// TIA Portal V18 export
// export: Created 2025-12-01T17:53:01.7250891Z, ExportSetting None, DisplayName Totally Integrated Automation Portal, DisplayVersion V18 Update 5, DisplayName TIA Portal Openness, DisplayVersion V18 Update 5, DisplayName TIA Portal Teamcenter Gateway, DisplayVersion V18, DisplayName TIA Portal Version Control Interface, DisplayVersion V18, DisplayName STEP 7 Professional, DisplayVersion V18 Update 5, DisplayName STEP 7 Safety, DisplayVersion V18, DisplayName WinCC Professional, DisplayVersion V18 Update 5
Screen "240_Cylinder_E1"  1280x800, Number=240, Template=02ManualUnit1
  ScreenLayer "Layer_0"
    FaceplateInstance "Cylinder_S71500_TP700_1" at 0,85 size 1279x80  FaceplateTypeName=03 FunctionBlocks@$@101 Cylinder@$@101.2 HMI@$@S7-1500@$@Cylinder_S71500_TP700 V 0.0.29
      Cy := STxxxCylinder011
      CylinderName := Cyl name
      HomeButtonName := Cyl go home button
      WorkButtonName := Cyl go work button
      HomeQaddress := Cyl home Q
      HomeIaddress := Cyl home I
      WorkIaddress := Cyl work I
      WorkQaddress := Cyl work Q
    Button "btnMenu4" at 384,725 size 128x75  StyleItem=BtnNormal20
    Button "btnMenu5" at 512,725 size 128x75  StyleItem=BtnNormal20
    Button "btnMenu6" at 640,725 size 128x75  StyleItem=BtnNormal20
    Button "btnMenu6_1" at 768,725 size 128x75  StyleItem=BtnNormal20
    Button "按钮_1" at 128,725 size 128x75  PictureOff=向右箭头_0, TextOff="E-气缸1 / E-Cylinder1", TextOn="E-气缸1 / E-Cylinder1"
      on Click: ActivateScreen(Screen name := , Object number := 0)
    Button "btnMenu4_1" at 256,725 size 128x75  TextOff="E-气缸2 / E-Cylinder2", TextOn="E-气缸2 / E-Cylinder2"
      on Click: ActivateScreen(Screen name := 246_Cylinder_E2, Object number := 0)
    GraphicView "图形视图_1" at 353,167 size 602x502  Picture=图形_52
    Button "btnMenu7" at 896,725 size 128x75
    Button "btnMenu7_1" at 1024,725 size 128x75
